FUNCTION_BLOCK FB_StateEnabled
VAR_IN_OUT
	stAxis  	: ARRAY [GVL.cXP .. GVL.cXM] OF ST_AxisGroup;
	bTopEntry	: BOOL;
END_VAR
VAR_INPUT
	eCommand			: E_Commands;
	stCalibrate			: ST_Calibrate;
	stChangeAxisEnable	: ST_ChangeAxisEnable;
	stChangeBrakeState	: ST_ChangeBrakeState;
	stClearAllFaults	: ST_ClearAllFaults;
	stClearAxisFaults	: ST_ClearAxisFaults;
	stCloseShutter		: ST_CloseShutter;
	stDisableAllAxes	: ST_DisableAllAxes;
	stEnableAllAxes		: ST_EnableAllAxes;
	stGoToProd			: ST_GoToProd;
	stHomeAxis			: ST_HomeAxis;
	stMoveAxisAbsolute	: ST_MoveAxisAbsolute;
	stMoveAxisRelative	: ST_MoveAxisRelative;
	stOpenShutter		: ST_OpenShutter;
	stReset				: ST_Reset;
	stTakeExposure		: ST_TakeExposure;
END_VAR
VAR_OUTPUT
	bCalibDone			: BOOL;
	bMotionDone			: BOOL;
	stOutCalibDone		: ST_CalibDone;
	stOutTimer			: ST_Timer;
	nSMState			: DINT;
END_VAR
VAR
	//state-machine
	eCurrentState	: E_StatesEnabled;
	eNextState		: E_StatesEnabled;
	fbMaint			: FB_StateMaint;
	fbProd			: FB_StateProd;
	bLowerEntry		: BOOL;
	
	//Event
	bIsCalibrated	: BOOL;
	bShutterReady	: BOOL;

	//Other var
	fbReset			: FB_Reset;
	bResetting		: BOOL;
	bResetEntry		: BOOL;
	bStopping		: BOOL;
	
END_VAR

(**)
IF bTopEntry = TRUE THEN
	bTopEntry := FALSE;
	(*Check if shutter blade sets are calibrated. If not, then go to still, otherwise go to previous state*)
	IF stAxis[GVL.cXP].bIsCalibrated AND stAxis[GVL.cXM].bIsCalibrated THEN
		eNextState := eCurrentState;
	ELSE
		eNextState := E_StatesEnabled.Maint;
	END_IF
END_IF	

IF eCurrentState <> eNextState THEN
	bLowerEntry := TRUE;
END_IF
eCurrentState := eNextState;

(* State Machine *)
CASE eCurrentState OF
	
	E_StatesEnabled.Maint:
		fbMaint(
			//inputs
			stAxis 				:= stAxis, 
			bTopEntry 			:= bLowerEntry, 
			eCommand			:= eCommand,
			stCalibrate			:= stCalibrate,
			stChangeAxisEnable	:= stChangeAxisEnable,
			stChangeBrakeState	:= stChangeBrakeState,
			stClearAllFaults	:= stClearAllFaults,
			stClearAxisFaults	:= stClearAxisFaults,
			stDisableAllAxes	:= stDisableAllAxes,
			stEnableAllAxes		:= stEnableAllAxes,
			stGoToProd			:= stGoToProd,
			stHomeAxis			:= stHomeAxis,
			stMoveAxisAbsolute	:= stMoveAxisAbsolute,
			stMoveAxisRelative	:= stMoveAxisRelative,
			//outputs
			bCalibDone			=> bCalibDone,
			bMotionDone			=> bMotionDone,
			stOutCalibDone		=> stOutCalibDone,
			nSMState			=> nSMState);	
		IF bShutterReady AND eCommand = E_Commands.goToProd THEN
			eNextState := E_StatesEnabled.Prod;
		END_IF
	
	E_StatesEnabled.Prod:
		fbProd(
			//inputs
			stAxis			:= stAxis, 
			bTopEntry 		:= bLowerEntry,
			eCommand		:= eCommand,
			fSpeed			:= stReset.speed,
			stOpenShutter	:= stOpenShutter,
			stCloseShutter	:= stCloseShutter,
			stTakeExposure	:= stTakeExposure,
			//outputs
			bMotionDone		=> bMotionDone,
			nSMState		=> nSMState,
			stOutTimer		=> stOutTimer);

END_CASE

//Reset routine
IF eCommand = E_Commands.reset THEN
	bResetting 	:= TRUE;
	bResetEntry	:= TRUE;
END_IF
IF bResetting THEN
	fbReset(stAxis:=stAxis, bResetEntry:=bResetEntry,bResetting:=bResetting,);
	eNextState := E_StatesEnabled.Maint;
	bLowerEntry := TRUE; //forces states in Maint to go to still state
END_IF


//Status for when shutter is ready to be put into prod mode.
bShutterReady := (stAxis[GVL.cXP].bBrake AND stAxis[GVL.cXM].bBrake) AND (stAxis[GVL.cXP].bIsCalibrated AND stAxis[GVL.cXM].bIsCalibrated) AND
	(
		((stAxis[GVL.cXP].axisRef.NcToPlc.ActPos<1) AND (stAxis[GVL.cXM].axisRef.NcToPlc.ActPos<1)) OR 
		((stAxis[GVL.cXP].axisRef.NcToPlc.ActPos>750) AND (stAxis[GVL.cXM].axisRef.NcToPlc.ActPos>750))
	);

END_FUNCTION_BLOCK

(* stored: Version 1.1.0.1, ProductVersion 3.1.4022.18
   POU FB_StateEnabled: Id {b94d2bdc-9aa0-4455-a0cd-476d7bce246d}, SpecialFunc None *)
